// TIA Portal project "FactoryIO_Template_S7-1200_V16_V16" (V16)
// Vorlageprojekt für das Buch mit Zielsystem S7-1200

(* hardware
DEVICE "S7-1200-Station_1"  S7-1200 Station
   slot 0: "Baugruppenträger_0"  Rack  V1.0
   slot 1: "PLC_1"  CPU 1211C DC/DC/DC  6ES7 211-1AE40-0XB0  V4.1
*)

// ===== PLC "PLC_1"  CPU 1211C DC/DC/DC =====

VAR_GLOBAL   // PLC tag table "Standard-Variablentabelle"
   "Start" AT %I0.0 : Bool;
   "Stop" AT %I0.1 : Bool;
   "Sensor 1" AT %I0.2 : Bool;
   "Sensor 2" AT %I0.3 : Bool;
   "Sensor 3" AT %I0.4 : Bool;
   "Sensor 4" AT %I0.5 : Bool;
   "Belt convyor(6m)" AT %Q0.0 : Bool;
   "Belt convyor(4m)1" AT %Q0.1 : Bool;
   "Belt convyor(4m)2" AT %Q0.2 : Bool;
   "Belt convyor(4m)3" AT %Q0.3 : Bool;
   "Pop Up Wheel Sorter 1(Right)(1)" AT %Q0.4 : Bool;
   "Pop Up Wheel Sorter 1(Left)(1)" AT %Q0.5 : Bool;
   "Pop Up Wheel Sorter 1(+)" AT %Q0.6 : Bool;
   "Start Button 1 (Light)" AT %Q0.7 : Bool;
   "StopButton 1 (Light)" AT %Q1.0 : Bool;
   "M1" AT %M0.0 : Bool;
   "M2" AT %M0.1 : Bool;
   "M3" AT %M0.2 : Bool;
   "M4" AT %M0.3 : Bool;
   "M5" AT %M0.4 : Bool;
   "M6" AT %M0.5 : Bool;
   "M7" AT %M0.6 : Bool;
   "M8" AT %M0.7 : Bool;
   "M9" AT %M1.0 : Bool;
   "M10" AT %M1.1 : Bool;
   "Tag_1" AT %M5.0 : Bool;
   "Tag_2" AT %M5.1 : Bool;
   "Tag_3" AT %M5.2 : Bool;
   "Tag_4" AT %M5.3 : Bool;
END_VAR

FUNCTION "MHJ-PLC-Lab-Function-S71200" : Void   // FC9000, SCL
{ S7_Optimized_Access := 'TRUE' }
VERSION : 0.1
   VAR_TEMP
      rdTimeReturn : Int;
      outputTime : DTL;
      SyncVal : Byte;
      forVal : Int;
      forVal_2 : Int;
      Value : Byte;
   END_VAR
   VAR CONSTANT
      CompVal : Byte := 16#34;
      Value_01 : Byte := 16#11;
      Value_01_DW : DWord := 16#A165_D992;
      Value_02_DW : DWord := 16#58BE_4401;
   END_VAR
BEGIN

   #Value:=PEEK(area := 16#82,
        dbNumber := 0,
        byteOffset := 511);
   #Value := #Value + 1;

   POKE(area := 16#82,
        dbNumber := 0,
        byteOffset := 511,
        value := #Value);

   POKE(area:=16#81,
        dbNumber:=0,
        byteOffset:=1016,
        value:=#Value_01_DW);
   POKE(area := 16#81,
        dbNumber := 0,
        byteOffset := 1020,
        value := #Value_02_DW);

   POKE(area := 16#81,
        dbNumber := 0,
        byteOffset := 511,
        value := B#16#00);

   FOR #forVal := 0 TO 120 DO
       FOR #forVal_2:=0 TO 10 DO
           #rdTimeReturn:=RD_SYS_T(#outputTime);
           #rdTimeReturn := WR_SYS_T(#outputTime);
           #rdTimeReturn := RD_SYS_T(#outputTime);
           #rdTimeReturn := WR_SYS_T(#outputTime);
       END_FOR;
       #SyncVal:= PEEK(area := 16#81,
                      dbNumber := 0,
                      byteOffset := 511);
       IF #SyncVal = #CompVal THEN
          GOTO M_1;
       END_IF;
   END_FOR;
   RETURN;

   M_1:
   POKE(area := 16#81,
        dbNumber := 0,
        byteOffset := 511,
        value := B#16#0);
END_FUNCTION

ORGANIZATION_BLOCK "Main"   // OB1, LAD, ProgramCycle
TITLE = "Main Program Sweep (Cycle)"
{ S7_Optimized_Access := 'TRUE' }
VERSION : 0.1
   VAR_INPUT
      Initial_Call : Bool;   // Initial call of this OB
      Remanence : Bool;   // =True, if remanent data are available
   END_VAR
   VAR_TEMP   // added for the SCL form of the ladder/FBD networks
      _w1 : Bool;
   END_VAR
BEGIN

REGION Network 1: Konnektierungsbaustein für PLC-Lab
   // Im Netzwerk 1 wird der Konnektierungsbaustein für PLC-Lab aufgerufen.
   // Dieser Aufruf darf nicht entfernt werden!
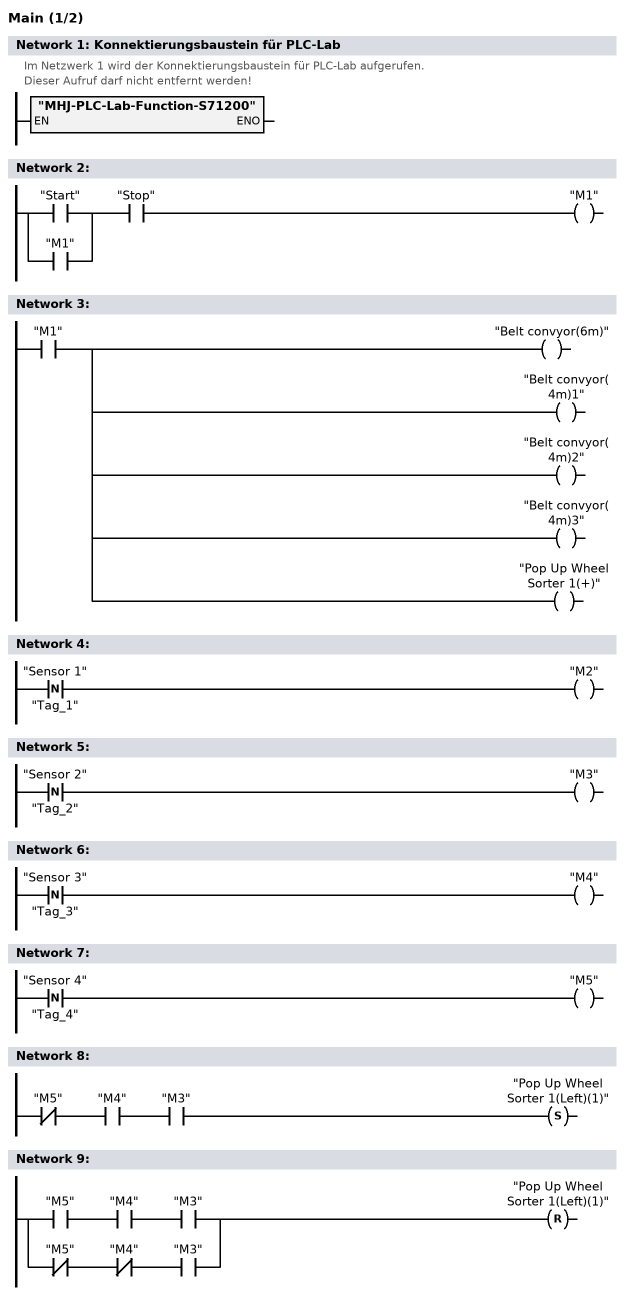
   RUNG wire#powerrail
      "MHJ-PLC-Lab-Function-S71200"()
   END_RUNG
   // the same network as SCL:
   "MHJ-PLC-Lab-Function-S71200"();
END_REGION

REGION Network 2
   RUNG wire#powerrail
      Contact( "Start" )
      wire#w1
      Contact( "Stop" )
      Coil( "M1" )
   END_RUNG
   RUNG wire#powerrail
      Contact( "M1" )
   END_RUNG wire#w1
   // the same network as SCL:
   "M1" := ("Start" OR "M1") AND "Stop";
END_REGION

REGION Network 3
   RUNG wire#powerrail
      Contact( "M1" )
      wire#w1
      Coil( "Belt convyor(6m)" )
   END_RUNG
   RUNG wire#w1
      Coil( "Belt convyor(4m)1" )
   END_RUNG
   RUNG wire#w1
      Coil( "Belt convyor(4m)2" )
   END_RUNG
   RUNG wire#w1
      Coil( "Belt convyor(4m)3" )
   END_RUNG
   RUNG wire#w1
      Coil( "Pop Up Wheel Sorter 1(+)" )
   END_RUNG
   // the same network as SCL:
   "Belt convyor(6m)" := "M1";
   "Belt convyor(4m)1" := "M1";
   "Belt convyor(4m)2" := "M1";
   "Belt convyor(4m)3" := "M1";
   "Pop Up Wheel Sorter 1(+)" := "M1";
END_REGION

REGION Network 4
   RUNG wire#powerrail
      N_Contact(operand := "Sensor 1", bit := "Tag_1")
      Coil( "M2" )
   END_RUNG
   // the same network as SCL:
   #_w1 := NOT "Sensor 1" AND "Tag_1";   // falling edge of "Sensor 1"
   "Tag_1" := "Sensor 1";
   "M2" := #_w1;
END_REGION

REGION Network 5
   RUNG wire#powerrail
      N_Contact(operand := "Sensor 2", bit := "Tag_2")
      Coil( "M3" )
   END_RUNG
   // the same network as SCL:
   #_w1 := NOT "Sensor 2" AND "Tag_2";   // falling edge of "Sensor 2"
   "Tag_2" := "Sensor 2";
   "M3" := #_w1;
END_REGION

REGION Network 6
   RUNG wire#powerrail
      N_Contact(operand := "Sensor 3", bit := "Tag_3")
      Coil( "M4" )
   END_RUNG
   // the same network as SCL:
   #_w1 := NOT "Sensor 3" AND "Tag_3";   // falling edge of "Sensor 3"
   "Tag_3" := "Sensor 3";
   "M4" := #_w1;
END_REGION

REGION Network 7
   RUNG wire#powerrail
      N_Contact(operand := "Sensor 4", bit := "Tag_4")
      Coil( "M5" )
   END_RUNG
   // the same network as SCL:
   #_w1 := NOT "Sensor 4" AND "Tag_4";   // falling edge of "Sensor 4"
   "Tag_4" := "Sensor 4";
   "M5" := #_w1;
END_REGION

REGION Network 8
   RUNG wire#powerrail
      I_Contact( "M5" )
      Contact( "M4" )
      Contact( "M3" )
      S_Coil( "Pop Up Wheel Sorter 1(Left)(1)" )
   END_RUNG
   // the same network as SCL:
   IF NOT "M5" AND "M4" AND "M3" THEN "Pop Up Wheel Sorter 1(Left)(1)" := TRUE; END_IF;
END_REGION

REGION Network 9
   RUNG wire#powerrail
      Contact( "M5" )
      Contact( "M4" )
      Contact( "M3" )
      wire#w1
      R_Coil( "Pop Up Wheel Sorter 1(Left)(1)" )
   END_RUNG
   RUNG wire#powerrail
      I_Contact( "M5" )
      I_Contact( "M4" )
      Contact( "M3" )
   END_RUNG wire#w1
   // the same network as SCL:
   IF ("M5" AND "M4" AND "M3") OR (NOT "M5" AND NOT "M4" AND "M3") THEN
       "Pop Up Wheel Sorter 1(Left)(1)" := FALSE;
   END_IF;
END_REGION

REGION Network 10
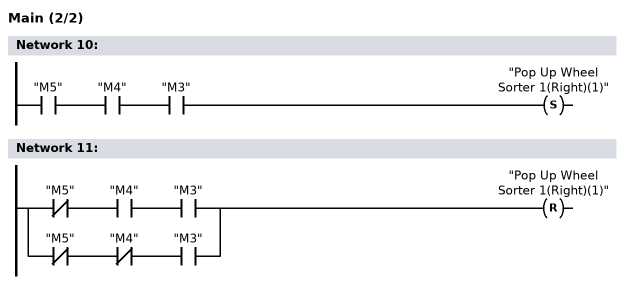
   RUNG wire#powerrail
      Contact( "M5" )
      Contact( "M4" )
      Contact( "M3" )
      S_Coil( "Pop Up Wheel Sorter 1(Right)(1)" )
   END_RUNG
   // the same network as SCL:
   IF "M5" AND "M4" AND "M3" THEN "Pop Up Wheel Sorter 1(Right)(1)" := TRUE; END_IF;
END_REGION

REGION Network 11
   RUNG wire#powerrail
      I_Contact( "M5" )
      Contact( "M4" )
      Contact( "M3" )
      wire#w1
      R_Coil( "Pop Up Wheel Sorter 1(Right)(1)" )
   END_RUNG
   RUNG wire#powerrail
      I_Contact( "M5" )
      I_Contact( "M4" )
      Contact( "M3" )
   END_RUNG wire#w1
   // the same network as SCL:
   IF (NOT "M5" AND "M4" AND "M3") OR (NOT "M5" AND NOT "M4" AND "M3") THEN
       "Pop Up Wheel Sorter 1(Right)(1)" := FALSE;
   END_IF;
END_REGION
END_ORGANIZATION_BLOCK